ABB RobotStudio station: IRB120 Parts Handling.rsstn

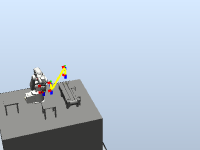
Station Station (saved by RobotStudio 6.8.8148.134)
Controller System1, task T_ROB1: task frame (RAPID world) sits at (0, 147.49, 949.54) mm in the station
Controller System1
  mechanical unit ROB_1: IRB120_3_58__01, 6 joints, base frame (0, 0, 0) mm
Layout (positions relative to the parent item):
  - IRB120_3_58__01 [mechanism, from Robots\IRB120_3_58_G_01.rslib] at (0, 147.49, 949.54) mm; joint values [-1.5004, 0.555, -0.6342, -0.0315, 1.6732, -1.4955] (rad or m)
  - 工作台 [part] at (0, 0, 518.6) mm, rotated rx 90 ry 0 rz 0 deg
  - Smart_Gripper_Servo_Fingers [mechanism] at (28.4, -287.7, 1490.75) mm, rotated rx 178.81 ry -1.9 rz 179.57 deg; joint values [0.025] (rad or m)
      TCP Servo at (0, 0, 114.2) mm
      links: HandBase, DownFinger, UpFinger, VacuumOne, VacuumTwo
  - 工件 [part] at (465.76, -304.56, 1137.86) mm
  - 传送带 [smart component]
      signals: DO do0
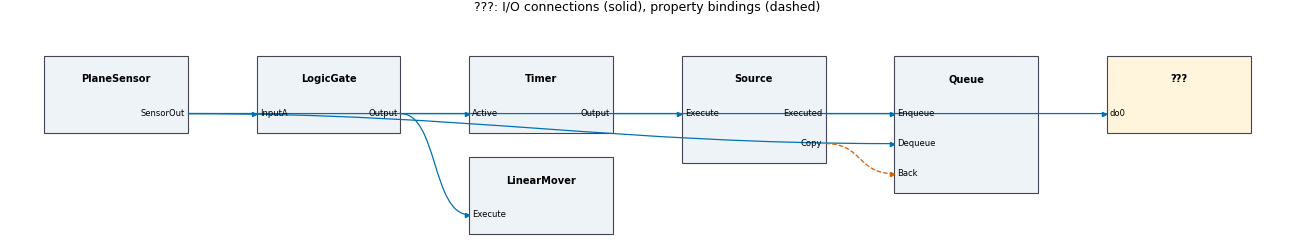
      connections:
        Timer.Output -> Source.Execute
        Source.Executed -> Queue.Enqueue
        PlaneSensor.SensorOut -> LogicGate.InputA
        LogicGate.Output -> Timer.Active
        LogicGate.Output -> LinearMover.Execute
        PlaneSensor.SensorOut -> Queue.Dequeue
        PlaneSensor.SensorOut -> 传送带.do0
        Source.Copy => Queue.Back
    - Timer [smart component, from Components\Timer.rslib]
        properties: StartTime=1; Interval=5; Repeat=true; CurrentTime=35.592
    - Source [smart component, from Components\Source.rslib]
        properties: Source=工件; Copy=(none); Parent=(none); Position=[0.465758 -0.304556 1.13786]; Orientation=[0 0 0]; Transient=false; PhysicsBehavior=0
    - Queue [smart component, from Components\Queue.rslib]
        properties: Back=(none); Front=(none); Queue={80330407-5a58-4c69-b2e3-bb833b888a4a};{9fb01dac-110b-452e-99c7-449fbd61bf52};{1fdbed24-73e7-4cdc-9659-c5dc2afe948c};{a4d3705a-74bf-4a3f-9169-404afb8702d5};{46bd0ae5-0552-4042-8276-f7110d3fe660};{10ceacc0-fe95-466c-99c0-06931470cbcc};{33f684c7-4ab7-4e3e-8fd4-209f09425ec2};{6ba75721-aefb-41b9-a23c-0a88ee2084a7};{fa522d1f-f0f5-4c87-924f-72403e0579d2}; NumberOfObjects=0
    - PlaneSensor [smart component, from Components\PlaneSensor.rslib]
        properties: Origin=[0.48521 0.163287 1.164314]; Axis1=[0 0 -0.02]; Axis2=[-0.04 0 0]; SensedPart=(none)
      - _sensorPart_ [part]
    - LogicGate [smart component, from Components\LogicGate.rslib]
        properties: Operator=NOT; Delay=0
    - LinearMover [smart component, from Components\LinearMover.rslib]
        properties: Object=Queue; Direction=[0 0.099 0]; Speed=0.1; Reference=Global; ReferenceObject=(none)
  - 夹爪 [smart component]
      signals: DI di0
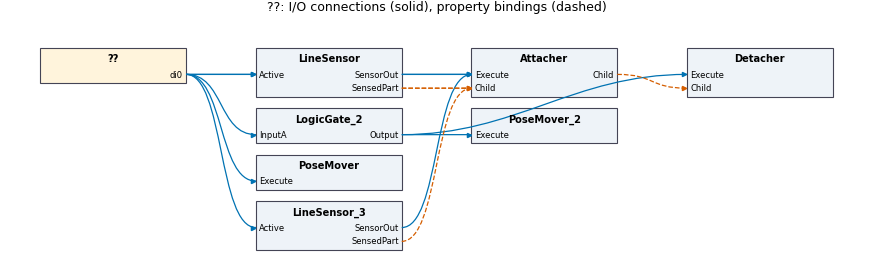
      connections:
        LineSensor.SensorOut -> Attacher.Execute
        LogicGate_2.Output -> Detacher.Execute
        夹爪.di0 -> LineSensor.Active
        夹爪.di0 -> LogicGate_2.InputA
        夹爪.di0 -> PoseMover.Execute
        LogicGate_2.Output -> PoseMover_2.Execute
        夹爪.di0 -> LineSensor_2.Active
        LineSensor_2.SensorOut -> Attacher.Execute
        夹爪.di0 -> LineSensor_3.Active
        LineSensor_3.SensorOut -> Attacher.Execute
        LineSensor.SensedPart => Attacher.Child
        Attacher.Child => Detacher.Child
        LineSensor_2.SensedPart => Attacher.Child
        LineSensor_3.SensedPart => Attacher.Child
    - Attacher [smart component, from Components\Attacher.rslib]
        properties: Parent=Smart_Gripper_Servo_Fingers; Flange=0; Child=(none); Mount=false; Offset=[0 0 0]; Orientation=[0 0 0]
    - Detacher [smart component, from Components\Detacher.rslib]
        properties: Child=(none); KeepPosition=true
    - LogicGate_2 [smart component, from Components\LogicGate.rslib]
        properties: Operator=NOT; Delay=0.1
    - PoseMover [smart component, from Components\PoseMover.rslib]
        properties: Mechanism=Smart_Gripper_Servo_Fingers; Pose=0; Duration=0
    - PoseMover_2 [smart component, from Components\PoseMover.rslib]
        properties: Mechanism=Smart_Gripper_Servo_Fingers; Pose=1; Duration=0
    - LineSensor_3 [smart component, from Components\LineSensor.rslib] at (-441.78, -436.7, 154.82) mm
        properties: Start=[0.467521 0.150698 1.255295]; End=[0.467521 0.150698 1.235295]; Radius=0.003; SensedPart=(none); SensedPoint=[0.0257441635131836 -0.286004638671875 1.25251879882813]
      - _sensorPart_ [part]
  - 写字台 [part] at (-560.7, 187.11, 1149.6) mm, rotated rx 90 ry 0 rz 0 deg
Attachment: Smart_Gripper_Servo_Fingers is attached to IRB120_3_58__01 / Link6
Attachment: LineSensor_3 is attached to Smart_Gripper_Servo_Fingers / HandBase
Station logic (signal -> signal, property => property):
  传送带.do0 -> System1.di00
  System1.do00 -> 夹爪.di0
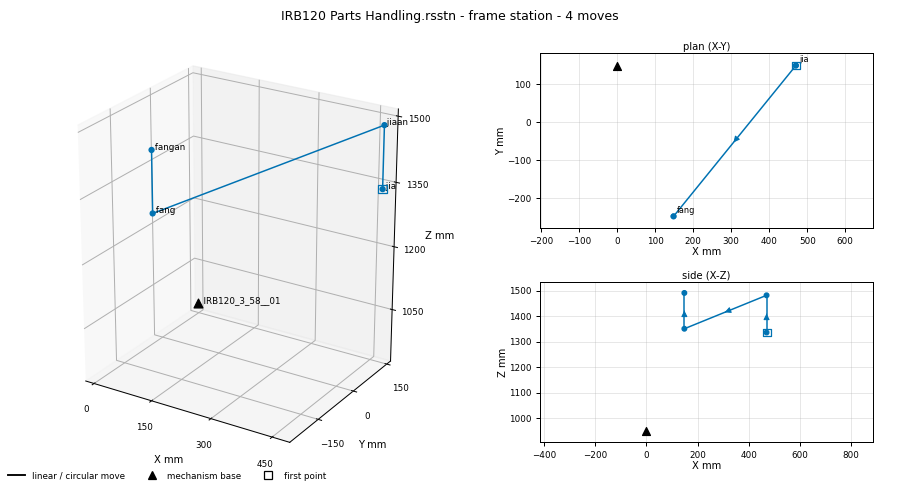
[picture p0: tool path of IRB120 Parts Handling.rsstn in frame station, 4 of 4 moves have a stored position in this frame; points joined in program order, loops and branches not executed]
Targets, tools, work objects and paths stored in the station, written as RAPID:
! task T_ROB1
MODULE CalibData
  PERS tooldata Servo:=[TRUE,[[0,0,114.2],[1,0,0,0]],[0.215,[8.7,12.3,49.2],[1,0,0,0],0.00021,0.00024,0.00009]];
ENDMODULE

! task T_ROB1
MODULE Module1
  CONST robtarget jia:=[[470.177984435,1.511223746,386.390605634],[0.016508173,-0.003881329,-0.999801768,-0.010432604],[0,0,0,0],[9E+09,9E+09,9E+09,9E+09,9E+09,9E+09]];
  CONST robtarget jiaan:=[[470.178016068,1.511223978,531.927787794],[0.016508193,-0.003881328,-0.999801768,-0.010432599],[0,0,0,0],[9E+09,9E+09,9E+09,9E+09,9E+09,9E+09]];
  CONST robtarget fang:=[[148.401105985,-395.19140183,401.049576169],[0.016508197,-0.003881289,-0.999801769,-0.010432567],[-1,-1,-1,0],[9E+09,9E+09,9E+09,9E+09,9E+09,9E+09]];
  CONST robtarget fangan:=[[148.401107386,-395.191406233,541.208958785],[0.016508189,-0.003881262,-0.999801769,-0.010432543],[-1,-1,-1,0],[9E+09,9E+09,9E+09,9E+09,9E+09,9E+09]];
  PROC Path_10()
    MoveL jia,v1000,z100,tool0\WObj:=wobj0;
    MoveL jiaan,v1000,z100,tool0\WObj:=wobj0;
    MoveL fang,v1000,z100,tool0\WObj:=wobj0;
    MoveL fangan,v1000,z100,tool0\WObj:=wobj0;
  ENDPROC
ENDMODULE

